// TIA Portal project "学习函数FC，分辨FC,FB的异同" (V16)

(* hardware
DEVICE "S7-1200 station_1"  S7-1200 Station
   slot 0: "Rack_0"  S7-1200 Rack  Rack  V1.0
   slot 1: "PLC_1"  CPU 1214C DC/DC/Rly  6ES7 214-1HG40-0XB0  V4.4
*)

// ===== PLC "PLC_1"  CPU 1214C DC/DC/Rly =====

VAR_GLOBAL   // PLC tag table "io"
   "启动信号" AT %I0.0 : Bool;
   "停止信号" AT %I0.1 : Bool;
   "复位信号" AT %I0.2 : Bool;
   "急停信号" AT %I0.3 : Bool;
   "左转到位i传感器" AT %I0.5 : Bool;
   "右转到位传感器" AT %I0.6 : Bool;
   "直行到位传感器" AT %I0.7 : Bool;
   "手动开关" AT %I1.0 : Bool;
   "自动开关" AT %I1.1 : Bool;
   "运行指示灯" AT %Q0.0 : Bool;
   "停止指示灯" AT %Q0.1 : Bool;
   "复位指示灯" AT %Q0.2 : Bool;
   "供料输送机" AT %Q0.3 : Bool;
   "直行电机" AT %Q0.4 : Bool;
   "左转电机" AT %Q0.5 : Bool;
   "右转电机" AT %Q0.6 : Bool;
   "产品原料分拣机" AT %Q0.7 : Bool;
   "产品基座分拣机" AT %Q1.0 : Bool;
   "产品盖分拣机" AT %Q1.1 : Bool;
   "物料生成器" AT %Q1.2 : Bool;
   "阻挡器" AT %Q1.3 : Bool;
   "视觉相机" AT %ID30 : DInt;
END_VAR

DATA_BLOCK "数据块_1"   // DB1
{ S7_Optimized_Access := 'TRUE' }
VERSION : 0.1
   VAR
      核心程序步 : Int;
      中间变量1 : Bool;
      中间变量2 : Bool;
      中间变量3 : Bool;
   END_VAR
BEGIN
END_DATA_BLOCK

FUNCTION "MHJ-PLC-Lab-Function-S71200" : Void   // FC9000, SCL
{ S7_Optimized_Access := 'TRUE' }
VERSION : 0.1
   VAR_TEMP
      rdTimeReturn : Int;
      outputTime : DTL;
      SyncVal : Byte;
      forVal : Int;
      forVal_2 : Int;
      Value : Byte;
   END_VAR
   VAR CONSTANT
      CompVal : Byte := 16#34;
      Value_01 : Byte := 16#11;
      Value_01_DW : DWord := 16#A165_D992;
      Value_02_DW : DWord := 16#58BE_4401;
   END_VAR
BEGIN

   #Value:=PEEK(area := 16#82,
        dbNumber := 0,
        byteOffset := 511);
   #Value := #Value + 1;

   POKE(area := 16#82,
        dbNumber := 0,
        byteOffset := 511,
        value := #Value);

   POKE(area:=16#81,
        dbNumber:=0,
        byteOffset:=1016,
        value:=#Value_01_DW);
   POKE(area := 16#81,
        dbNumber := 0,
        byteOffset := 1020,
        value := #Value_02_DW);

   POKE(area := 16#81,
        dbNumber := 0,
        byteOffset := 511,
        value := B#16#00);

   FOR #forVal := 0 TO 120 DO
       FOR #forVal_2:=0 TO 10 DO
           #rdTimeReturn:=RD_SYS_T(#outputTime);
           #rdTimeReturn := WR_SYS_T(#outputTime);
           #rdTimeReturn := RD_SYS_T(#outputTime);
           #rdTimeReturn := WR_SYS_T(#outputTime);
       END_FOR;
       #SyncVal:= PEEK(area := 16#81,
                      dbNumber := 0,
                      byteOffset := 511);
       IF #SyncVal = #CompVal THEN
          GOTO M_1;
       END_IF;
   END_FOR;
   RETURN;

   M_1:
   POKE(area := 16#81,
        dbNumber := 0,
        byteOffset := 511,
        value := B#16#0);
END_FUNCTION

ORGANIZATION_BLOCK "Main"   // OB1, LAD, ProgramCycle
TITLE = "Main Program Sweep (Cycle)"
{ S7_Optimized_Access := 'TRUE' }
VERSION : 0.1
   VAR_INPUT
      Initial_Call : Bool;   // Initial call of this OB
      Remanence : Bool;   // =True, if remanent data are available
   END_VAR
   VAR_TEMP   // added for the SCL form of the ladder/FBD networks
      _w1 : Bool;
   END_VAR
BEGIN

REGION Network 1
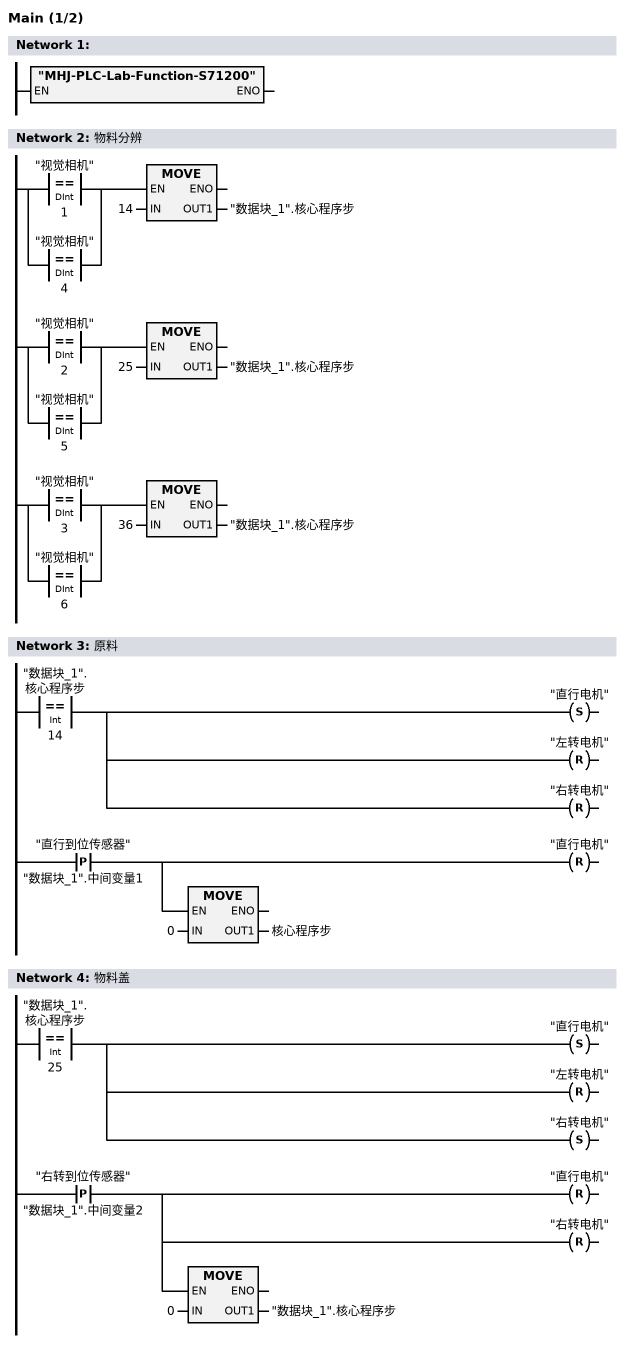
   RUNG wire#powerrail
      "MHJ-PLC-Lab-Function-S71200"()
   END_RUNG
   // the same network as SCL:
   "MHJ-PLC-Lab-Function-S71200"();
END_REGION

REGION Network 2: 物料分辨
   RUNG wire#powerrail
      { S7_Templates := "SrcType := DInt" } EQ_Contact(in1 := "视觉相机", in2 := 1)
      wire#w1
      Move(in := 14, out1 => "数据块_1".核心程序步)
   END_RUNG
   RUNG wire#powerrail
      { S7_Templates := "SrcType := DInt" } EQ_Contact(in1 := "视觉相机", in2 := 4)
   END_RUNG wire#w1
   RUNG wire#powerrail
      { S7_Templates := "SrcType := DInt" } EQ_Contact(in1 := "视觉相机", in2 := 2)
      wire#w2
      Move(in := 25, out1 => "数据块_1".核心程序步)
   END_RUNG
   RUNG wire#powerrail
      { S7_Templates := "SrcType := DInt" } EQ_Contact(in1 := "视觉相机", in2 := 5)
   END_RUNG wire#w2
   RUNG wire#powerrail
      { S7_Templates := "SrcType := DInt" } EQ_Contact(in1 := "视觉相机", in2 := 3)
      wire#w3
      Move(in := 36, out1 => "数据块_1".核心程序步)
   END_RUNG
   RUNG wire#powerrail
      { S7_Templates := "SrcType := DInt" } EQ_Contact(in1 := "视觉相机", in2 := 6)
   END_RUNG wire#w3
   // the same network as SCL:
   IF ("视觉相机" = 1) OR ("视觉相机" = 4) THEN "数据块_1".核心程序步 := 14; END_IF;
   IF ("视觉相机" = 2) OR ("视觉相机" = 5) THEN "数据块_1".核心程序步 := 25; END_IF;
   IF ("视觉相机" = 3) OR ("视觉相机" = 6) THEN "数据块_1".核心程序步 := 36; END_IF;
END_REGION

REGION Network 3: 原料
   RUNG wire#powerrail
      { S7_Templates := "SrcType := Int" } EQ_Contact(in1 := "数据块_1".核心程序步, in2 := 14)
      wire#w1
      S_Coil( "直行电机" )
   END_RUNG
   RUNG wire#w1
      R_Coil( "左转电机" )
   END_RUNG
   RUNG wire#w1
      R_Coil( "右转电机" )
   END_RUNG
   RUNG wire#powerrail
      P_Contact(operand := "直行到位传感器", bit := "数据块_1".中间变量1)
      wire#w2
      R_Coil( "直行电机" )
   END_RUNG
   RUNG wire#w2
      Move(in := 0, out1 => 核心程序步)
   END_RUNG
   // the same network as SCL:
   IF "数据块_1".核心程序步 = 14 THEN
       "直行电机" := TRUE;
       "左转电机" := FALSE;
       "右转电机" := FALSE;
   END_IF;
   #_w1 := "直行到位传感器" AND NOT "数据块_1".中间变量1;   // rising edge of "直行到位传感器"
   "数据块_1".中间变量1 := "直行到位传感器";
   IF #_w1 THEN
       "直行电机" := FALSE;
       核心程序步 := 0;
   END_IF;
END_REGION

REGION Network 4: 物料盖
   RUNG wire#powerrail
      { S7_Templates := "SrcType := Int" } EQ_Contact(in1 := "数据块_1".核心程序步, in2 := 25)
      wire#w1
      S_Coil( "直行电机" )
   END_RUNG
   RUNG wire#w1
      R_Coil( "左转电机" )
   END_RUNG
   RUNG wire#w1
      S_Coil( "右转电机" )
   END_RUNG
   RUNG wire#powerrail
      P_Contact(operand := "右转到位传感器", bit := "数据块_1".中间变量2)
      wire#w2
      R_Coil( "直行电机" )
   END_RUNG
   RUNG wire#w2
      R_Coil( "右转电机" )
   END_RUNG
   RUNG wire#w2
      Move(in := 0, out1 => "数据块_1".核心程序步)
   END_RUNG
   // the same network as SCL:
   IF "数据块_1".核心程序步 = 25 THEN
       "直行电机" := TRUE;
       "左转电机" := FALSE;
       "右转电机" := TRUE;
   END_IF;
   #_w1 := "右转到位传感器" AND NOT "数据块_1".中间变量2;   // rising edge of "右转到位传感器"
   "数据块_1".中间变量2 := "右转到位传感器";
   IF #_w1 THEN
       "直行电机" := FALSE;
       "右转电机" := FALSE;
       "数据块_1".核心程序步 := 0;
   END_IF;
END_REGION

REGION Network 5: 物料基座
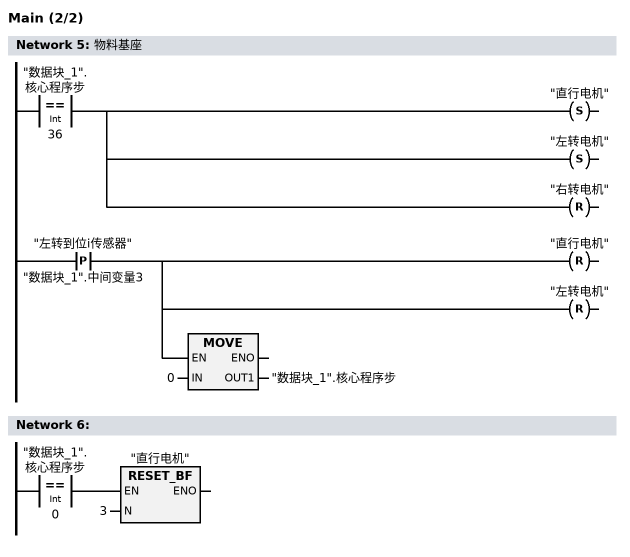
   RUNG wire#powerrail
      { S7_Templates := "SrcType := Int" } EQ_Contact(in1 := "数据块_1".核心程序步, in2 := 36)
      wire#w1
      S_Coil( "直行电机" )
   END_RUNG
   RUNG wire#w1
      S_Coil( "左转电机" )
   END_RUNG
   RUNG wire#w1
      R_Coil( "右转电机" )
   END_RUNG
   RUNG wire#powerrail
      P_Contact(operand := "左转到位i传感器", bit := "数据块_1".中间变量3)
      wire#w2
      R_Coil( "直行电机" )
   END_RUNG
   RUNG wire#w2
      R_Coil( "左转电机" )
   END_RUNG
   RUNG wire#w2
      Move(in := 0, out1 => "数据块_1".核心程序步)
   END_RUNG
   // the same network as SCL:
   IF "数据块_1".核心程序步 = 36 THEN
       "直行电机" := TRUE;
       "左转电机" := TRUE;
       "右转电机" := FALSE;
   END_IF;
   #_w1 := "左转到位i传感器" AND NOT "数据块_1".中间变量3;   // rising edge of "左转到位i传感器"
   "数据块_1".中间变量3 := "左转到位i传感器";
   IF #_w1 THEN
       "直行电机" := FALSE;
       "左转电机" := FALSE;
       "数据块_1".核心程序步 := 0;
   END_IF;
END_REGION

REGION Network 6
   // no SCL statement known for RBitfield: written as a call
   IF "数据块_1".核心程序步 = 0 THEN RESET_BF(operand := "直行电机", n := 3); END_IF;
END_REGION
END_ORGANIZATION_BLOCK